FUNCTION F_SAFETY_StatusFB_TO_AND 	: ST_SAFETY_FBAND 		(* Struktura dedykowana *)
VAR_INPUT
	stFBStatus						: ST_SAFETY_FBStatus; 	(* Struktura ogolna *)
END_VAR

F_SAFETY_StatusFB_TO_AND.uStatus.stStatusWords 		:= stFBStatus;									(* Przepisanie *)
F_SAFETY_StatusFB_TO_AND.eState					 	:= stFBStatus.BState;							(* Ustawienie enum *)

END_FUNCTION

(* stored: Version 1.1.0.1, ProductVersion 3.1.4022.12
   POU F_SAFETY_StatusFB_TO_AND: Id {ffab16de-166b-4c20-8f70-03be8dae869d}, SpecialFunc None *)
